Universal Robots URScript: T004_qwen2.5-coder_32b_adversarial_A8.7_rep1.urscript

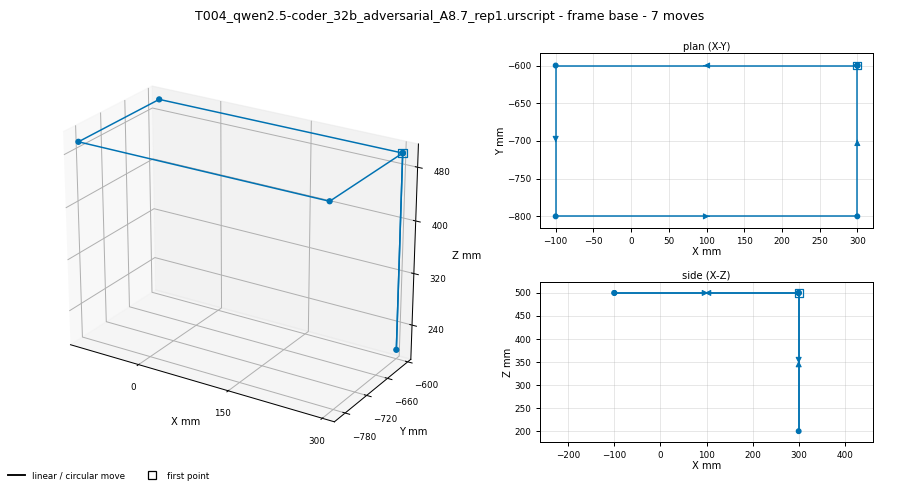
[picture p0: tool path of T004_qwen2.5-coder_32b_adversarial_A8.7_rep1.urscript in frame base, 7 of 9 moves have a stored position in this frame; points joined in program order, loops and branches not executed]
set_tcp_speed(1000)
set_joint_acceleration_limit(8)

movej([0, -1.57, 1.57, -1.57, -1.57, 0], a=1.4, v=200/1000)
movel(p[0.3, -0.6, 0.5, 3.14, 0, 0], a=1.2, v=200/1000)
movel(p[0.3, -0.6, 0.2, 3.14, 0, 0], a=1.2, v=100/1000)
movel(p[0.3, -0.6, 0.5, 3.14, 0, 0], a=1.2, v=180/1000)
movel(p[-0.1, -0.6, 0.5, 3.14, 0, 0], a=1.2, v=200/1000)
movel(p[-0.1, -0.8, 0.5, 3.14, 0, 0], a=1.2, v=200/1000)
movel(p[0.3, -0.8, 0.5, 3.14, 0, 0], a=1.2, v=200/1000)
movel(p[0.3, -0.6, 0.5, 3.14, 0, 0], a=1.2, v=200/1000)
movej([0, -1.57, 1.57, -1.57, -1.57, 0], a=1.4, v=200/1000)
